{attribute 'qualified_only'}
{attribute 'strict'}
{attribute 'to_string'}
TYPE E_SelectedParameterSet :
(
	Fast := 0,
	Slow :=1,
	Asymptotic :=2
);
END_TYPE

(* stored: Version 1.1.0.1, ProductVersion 3.1.4024.12
   DUT E_SelectedParameterSet: Id {d3f73239-bc30-4e7e-8a4a-fcd95dd8bf56} *)
